Staubli VAL3: selectedCheck.pgx

program selectedCheck()
begin
  if bSelectedItems[0]==true and bSelectedItems[1]==true and bSelectedItems[2]==true and bSelectedItems[3]==true and bSelectedItems[4]==true and bSelectedItems[5]==true
    bSelectItem = false
  else
    bSelectItem = true
  endIf

end
